// TIA Portal V17 export
// export: Created 2024-09-15T12:30:21.3696437Z, ExportSetting WithDefaults, DisplayName Totally Integrated Automation Portal, DisplayVersion V17, DisplayName TIA Portal Openness, DisplayVersion V17, DisplayName TIA Portal Version Control Interface, DisplayVersion V17, DisplayName STEP 7 Professional, DisplayVersion V17, DisplayName STEP 7 Safety, DisplayVersion V17, DisplayName WinCC Professional, DisplayVersion V17
VAR_GLOBAL   // PLC tag table "SLD - Sorting Line with Detection"
   IX_SLD_PulseCounter_I1 AT %I3.0 : Bool;   // SLD - I1 = Pulse counter   {ExternalAccessible false, ExternalVisible false, ExternalWritable false}
   IX_SLD_LightBarrierInlet_I2 AT %I3.1 : Bool;   // SLD - I2 = Light barrier inlet   {ExternalAccessible false, ExternalVisible false, ExternalWritable false}
   IX_SLD_LightBarrierBehindColorSensor_I3 AT %I3.2 : Bool;   // SLD - I3 = Light barrier behind color sensor   {ExternalAccessible false, ExternalVisible false, ExternalWritable false}
   IW_SLD_ColorSensor_A4 AT %IW7 : Word;   // SLD - A4 = Color sensor   {ExternalAccessible false, ExternalVisible false, ExternalWritable false}
   IX_SLD_LightBarrierWhite_I5 AT %I3.3 : Bool;   // SLD - I5 = Light barrier white   {ExternalAccessible false, ExternalVisible false, ExternalWritable false}
   IX_SLD_LightBarrierRed_I6 AT %I3.4 : Bool;   // SLD - I6 = Light barrier red   {ExternalAccessible false, ExternalVisible false, ExternalWritable false}
   IX_SLD_LightBarrierBlue_I7 AT %I3.5 : Bool;   // SLD - I7 = Light barrier blue   {ExternalAccessible false, ExternalVisible false, ExternalWritable false}
   QX_SLD_M1_ConveyorBelt_Q1 AT %Q5.0 : Bool;   // SLD - Q1 = Motor M1conveyor belt   {ExternalAccessible false, ExternalVisible false, ExternalWritable false}
   QX_SLD_Compressor_Q2 AT %Q5.1 : Bool;   // SLD - Q2 = Compressor   {ExternalAccessible false, ExternalVisible false, ExternalWritable false}
   QX_SLD_ValveFirstEjectorWhite_Q3 AT %Q5.2 : Bool;   // SLD - Q3 = Valve first ejector (white)   {ExternalAccessible false, ExternalVisible false, ExternalWritable false}
   QX_SLD_ValveSecondEjectorRed_Q4 AT %Q5.3 : Bool;   // SLD - Q4 = Valve second ejector (red)   {ExternalAccessible false, ExternalVisible false, ExternalWritable false}
   QX_SLD_ValveThirdEjectorBlue_Q5 AT %Q5.4 : Bool;   // SLD - Q5 = Valve third ejector (blue)   {ExternalAccessible false, ExternalVisible false, ExternalWritable false}
END_VAR
